// Annex I I.3 - jog frame for manual motion. Manual only, release-gated (S7.6).
{attribute 'qualified_only'}
TYPE E_JogMode :
(
    JOINT     := 0,
    CARTESIAN := 1,
    TOOL      := 2
) DINT;
END_TYPE

(* stored: Version 1.1.0.1, ProductVersion 3.1.4024.12
   DUT E_JogMode: Id {65611445-9828-453d-9b11-9f93a32b0988} *)
